TYPE ST_StateHistory :
STRUCT
	state		: INT;
	stateTime	: TIME;
	ts			: TIMESTRUCT;
END_STRUCT
END_TYPE

(* stored: Version 1.1.0.1, ProductVersion 3.1.4024.10
   DUT ST_StateHistory: Id {d47ab69b-df99-412d-bb10-99fbd65e3269} *)
